(* IEC 61131-3 sources: volt/packages/volt-lsp-iec/test-corpus/pro2193/Device/Plc Logic/Application/03 Hardware Units/31 SER/31.11 - Magazines/Motors/Drawer Magazine/Interfaces %2F Data, 4 files *)

(* ---- MagazineMotors_Drawer_BrinkData.dut ---- *)
TYPE MagazineMotors_Drawer_BrinkData :
STRUCT
	lrJerk			: LREAL;																	// Maximum jerk					(m/s³ or °/s³)
	rRefPos			: ARRAY[PickPlaceAxesNames.A1..PickPlaceAxesNames.A2] OF REAL;				// Position on reference point	(mm or °)
	rSWLimitPos		: ARRAY[PickPlaceAxesNames.A1..PickPlaceAxesNames.A2] OF REAL	:= [500.0];		// Positive software limit		(mm or °)
	rSWLimitNeg		: ARRAY[PickPlaceAxesNames.A1..PickPlaceAxesNames.A2] OF REAL	:= [-1.0];		// Negative software limit		(mm or °)
	rSWLimitPos_Z	: REAL	:= 1500;															// Positive software limit of virtual Z axis		(mm or °)
	rSWLimitNeg_Z	: REAL	:= 700;																// Negative software limit of virtual Z axis		(mm or °)
END_STRUCT
END_TYPE

(* ---- MagazineMotors_Drawer_Data.dut ---- *)
TYPE MagazineMotors_Drawer_Data :
STRUCT
	waitingPos				: PositionWithLimitsType;	// Position where to wait for the inlay-core (in case of wrap labels)
	labelTakeOverPos		: PositionWithLimitsType;	// Position where to give the labels to the Xi-axis

	getNewLabelsUpperPos	: PositionWithLimitsType;	// Position where to take-out new label from the stockpile in the upper drawer
	getNewLabelsLowerPos	: PositionWithLimitsType;	// Position where to take-out new label from the stockpile in the lower drawer

	DistanceSlowUpFromLabel		: REAL;					// Distance slow movement from label pickup after taking the labels
	VelocitySlowUpFromLabel		: REAL;					// Velocity [m/s]
	SafeDistanceAboveDrawers	: REAL;					// Distance above the drawers where it is safe to go to takeover position

	ProfileMovingDown			: ProfileType;
	ProfileMovingUp				: ProfileType;
	ProfileWaitingToTakeover	: ProfileType;
END_STRUCT
END_TYPE

(* ---- IMagazineMotors_Drawer_Commands.itf ---- *)
// Commands specific for a Magazine Unit
INTERFACE IMagazineMotors_Drawer_Commands
EXTENDS IModuleBase, IModuleManualControlEnabled, IModuleStartCommand, IModuleHasSafePos

// Returns true if the motor is in the required position
METHOD PUBLIC InPositionAt : BOOL
VAR_INPUT
	position	: MagazineMotors_Positions;
	tolerance	: REAL;
END_VAR

END_METHOD

METHOD ProfileHomeToSafePosition : BOOL

END_METHOD

METHOD ProfileSafeDistanceAboveDrawer : BOOL
VAR_INPUT
	drawer	: enumDrawer;
END_VAR

END_METHOD

METHOD ProfileToHorizontal : BOOL
VAR_INPUT
	drawer	: enumDrawer;
END_VAR

END_METHOD

// Move to any position that is vertical. For example  Waiting -> Takeover or Drawer -> Waiting
METHOD ProfileToVertical : BOOL
VAR_INPUT
	drawer		: enumDrawer;
	endPosition	: MagazineMotors_Positions;	// Should be any position where arm is vertical (so to transfer a label to Xi)
END_VAR

END_METHOD

// Command to reset the module. Servodrives are homed.
METHOD PUBLIC Reset : BOOL	// Returns true when homing done

END_METHOD

END_INTERFACE

(* ---- KinematicModelFB.pou ---- *)
FUNCTION_BLOCK KinematicModelFB
EXTENDS L_MC4P_Kin_Ref_Generic
VAR_INPUT
	lrArmLength : LREAL := 895;
END_VAR
VAR_OUTPUT
END_VAR
VAR
END_VAR
VAR CONSTANT
	Deg90ToRads : LREAL := 1.5707963267949; // Radians value for 90 degrees
END_VAR

%LANGUAGE ST

END_FUNCTION_BLOCK

METHOD CalcBackwardTrafo : WORD
VAR_IN_OUT
	AxesGroup		: L_MC4P.AXES_GROUP_KIN;
	alrPosFlange	: ARRAY[1..6] OF LREAL;
	alrPosAxes		: ARRAY[1..6] OF LREAL;
	aiConfiguration	: ARRAY[1..6] OF INT;
END_VAR
VAR_INST
	actualXPos			: LREAL;
END_VAR

%LANGUAGE ST
// Implement here: Backward-Trafo / inverse kinematics:
// Calculate the ACS-Positions according to position of the flange (TCS-Position, defined in MCS)

IF alrPosFlange[1] > lrArmLength THEN
	actualXPos		:= lrArmLength - (alrPosFlange[1] - lrArmLength);
	alrPosAxes[1]	:= alrPosFlange[3] - SQRT(EXPT(lrArmLength, 2) - EXPT(lrArmLength - actualXPos,2));
	alrPosAxes[2]	:= alrPosFlange[3] + SQRT(EXPT(lrArmLength, 2) - EXPT(actualXPos, 2));

ELSIF alrPosFlange[1] < 0 THEN
	actualXPos		:= ABS(alrPosFlange[1]);
	alrPosAxes[1]	:= alrPosFlange[3] + SQRT(EXPT(lrArmLength, 2) - EXPT(lrArmLength - actualXPos,2));
	alrPosAxes[2]	:= alrPosFlange[3] - SQRT(EXPT(lrArmLength, 2) - EXPT(actualXPos, 2));

ELSE

	actualXPos		:= alrPosFlange[1];
	alrPosAxes[1]	:= alrPosFlange[3] - SQRT(EXPT(lrArmLength, 2) - EXPT(lrArmLength - actualXPos,2));		// This is the calculated position of the M1-axis
	alrPosAxes[2]	:= alrPosFlange[3] - SQRT(EXPT(lrArmLength, 2) - EXPT(actualXPos, 2));					// This is the calculated position of the M2-axis
END_IF

END_METHOD

METHOD CalcForwardTrafo : WORD
VAR_IN_OUT
	AxesGroup		: L_MC4P.AXES_GROUP_KIN;
	alrPosFlange	: ARRAY[1..6] OF LREAL;
	alrPosAxes		: ARRAY[1..6] OF LREAL;
END_VAR
VAR_INST
	diffAxes		: LREAL;
	diffAngle		: LREAL;
	diffAngleDeg	: LREAL;
	distAxes		: LREAL;
	angleA1			: LREAL;
	actualXPos		: LREAL;
END_VAR

%LANGUAGE ST
// Implement here: Forward-Trafo / direct kinematics:
// Calculate the position of the flange (TCS-Position, defined in MCS) according to ACS-Positions

// Difference between the Axis positions
diffAxes		:= alrPosAxes[1] - alrPosAxes[2];

// Angle in radians of the line between the Axis positions referred to the horizontal line
diffAngle		:= ATAN(diffAxes / lrArmLength);

// Length of the line between the Axis positions
distAxes		:= SQRT(EXPT(lrArmLength, 2) + EXPT(diffAxes, 2));

// Angle in radians of the gripper measured to the vertical line
angleA1			:= Deg90ToRads - diffAngle - ACOS((distAxes / 2) / lrArmLength);

// Real actual X-position
actualXPos		:=  SIN(angleA1) * lrArmLength;

// Angle in degrees
diffAngleDeg	:= diffAngle * 180.0 / GVL_Constants.pi;

// X position was at maximum of 895, and went back again. Make 'virtual' X position > lrArmLength
IF diffAngleDeg < -45 THEN
	alrPosFlange[1]	:= (lrArmLength - actualXPos) + lrArmLength;											// X-position
	alrPosFlange[3]	:= SQRT(EXPT(lrArmLength, 2) - EXPT((lrArmLength - actualXPos), 2)) + alrPosAxes[1];	// Z-position

// X position was at minimum of 0, and went back again. Make 'virtual' X position < 0
ELSIF diffAngleDeg > 45 THEN
	alrPosFlange[1]	:= -actualXPos;																			// X-position
	alrPosFlange[3]	:= SQRT(EXPT(lrArmLength, 2) - EXPT((actualXPos), 2)) + alrPosAxes[2];					// Z-position

// X position is within normal operating range
ELSE
	alrPosFlange[1]	:= actualXPos;																			// X-position
	alrPosFlange[3]	:= SQRT(EXPT(lrArmLength, 2) - EXPT((lrArmLength - actualXPos), 2)) + alrPosAxes[1];	// Z-position
END_IF

END_METHOD

METHOD CalculateConfiguration : WORD
VAR_IN_OUT
	AxesGroup	: L_MC4P.AXES_GROUP_KIN;
	alrPosFlange	: ARRAY[1..6] OF LREAL;
	alrPosAxes	: ARRAY[1..6] OF LREAL;
	aiConfiguration	: ARRAY[1..6] OF INT;
END_VAR

%LANGUAGE ST
// Use this method, if your Backwardtransformation has more than one solution, depending on the actual position of the ACS-Axes

END_METHOD

METHOD CalculateParameter

%LANGUAGE ST
// Calculate variables depending on user-defined parameters

END_METHOD

METHOD CheckParameter : BOOL

%LANGUAGE ST
CheckParameter := TRUE;
END_METHOD

METHOD SetACSAxisType
// Overwrite this method, if ACS-axes in user-trafo are different from the default implementation
VAR_OUTPUT CONSTANT
	aeAxes: ARRAY[1..6] OF L_MC4P_AxisType := [L_MC4P_AxisType.linear,
											   L_MC4P_AxisType.linear,
											   L_MC4P_AxisType.unconnected,
											   L_MC4P_AxisType.unconnected,
											   L_MC4P_AxisType.unconnected,
											   L_MC4P_AxisType.unconnected];
END_VAR

%LANGUAGE ST
END_METHOD
